FUNCTION_BLOCK INFLUX_DB_2
  {SET_ATTRIBUTE(OpcUa, POINT.ENDPOINT)}
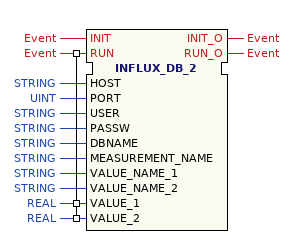
  EVENT_INPUT
    INIT;
    RUN WITH VALUE_1, VALUE_2;
  END_EVENT
  EVENT_OUTPUT
    INIT_O;
    RUN_O;
  END_EVENT
  VAR_INPUT
    HOST : STRING; {SET_ATTRIBUTE(OpcUa, Constant)}
    PORT : UINT; {SET_ATTRIBUTE(OpcUa, Constant)}
    USER : STRING; {SET_ATTRIBUTE(OpcUa, Constant)}
    PASSW : STRING; {SET_ATTRIBUTE(OpcUa, Constant)}
    DBNAME : STRING; {SET_ATTRIBUTE(OpcUa, Constant)}
    MEASUREMENT_NAME : STRING; {SET_ATTRIBUTE(OpcUa, Constant)}
    VALUE_NAME_1 : STRING; {SET_ATTRIBUTE(OpcUa, Constant)}
    VALUE_NAME_2 : STRING; {SET_ATTRIBUTE(OpcUa, Constant)}
    VALUE_1 : REAL; {SET_ATTRIBUTE(OpcUa, Variable)}
    VALUE_2 : REAL; {SET_ATTRIBUTE(OpcUa, Variable)}
  END_VAR
END_FUNCTION_BLOCK
